// TIA Portal V17 export
// export: Created 2024-09-02T21:27:54.0688981Z, ExportSetting WithDefaults, DisplayName Totally Integrated Automation Portal, DisplayVersion V17 Update 7, DisplayName TIA Portal Openness, DisplayVersion V17 Update 7, DisplayName TIA Portal Version Control Interface, DisplayVersion V17, DisplayName SINAMICS Startdrive Advanced, DisplayVersion V17 SP2, DisplayName SINAMICS Startdrive G110M, G120, G120C, G120D, G120P, G115D, DisplayVersion V17 SP2, DisplayName SINAMICS Startdrive G130, G150, S120, S150, SINAMICS MV, S210, DisplayVersion V17 SP2, DisplayName STEP 7 Professional, DisplayVersion V17 Update 7, DisplayName STEP 7 Safety, DisplayVersion V17 Update 6, DisplayName WinCC Advanced / Unified PC, DisplayVersion V17 Update 7
FUNCTION "inputsMapping" : Void   // FC1, LAD
{ S7_Optimized_Access := 'TRUE' }
VERSION : 0.1
// stored: AutoNumber true, IsIECCheckEnabled false, SetENOAutomatically false, UDAEnableTagReadback false
BEGIN

REGION Network 1: A00.- Clear Data
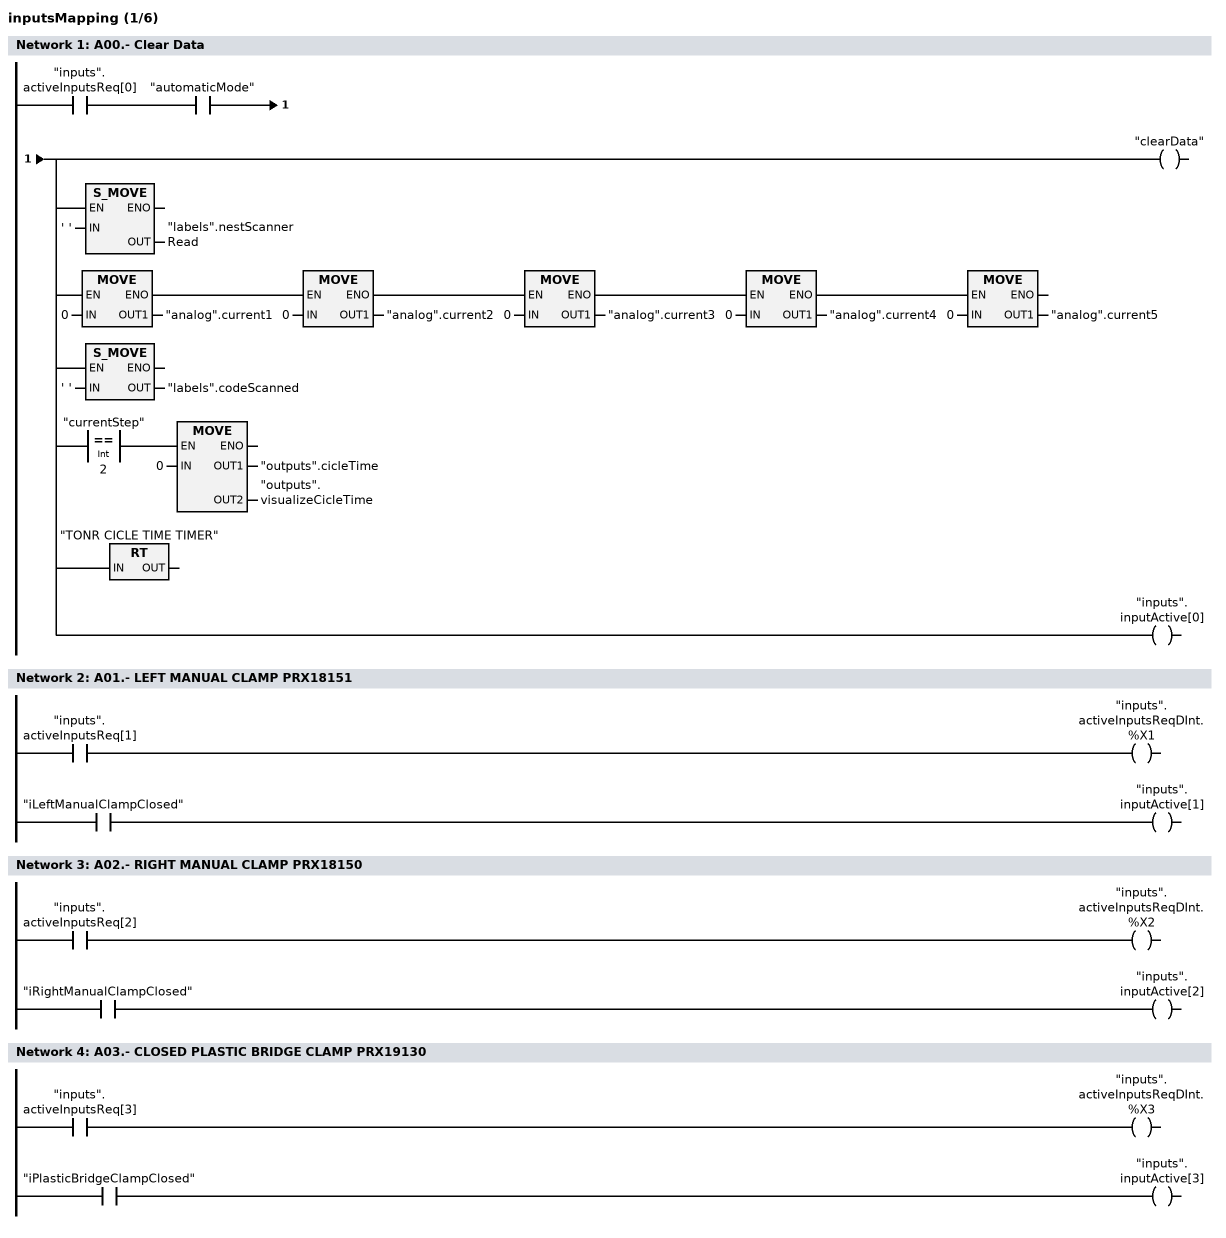
   RUNG wire#powerrail
      Contact( "inputs".activeInputsReq[0] )
      Contact( "automaticMode" )
      wire#w1
      Coil( "clearData" )
   END_RUNG
   RUNG wire#w1
      S_Move(in := ' ', out => "labels".nestScannerRead)
   END_RUNG
   RUNG wire#w1
      Move(in := 0, out1 => "analog".current1)
      Move(in := 0, out1 => "analog".current2)
      Move(in := 0, out1 => "analog".current3)
      Move(in := 0, out1 => "analog".current4)
      Move(in := 0, out1 => "analog".current5)
   END_RUNG
   RUNG wire#w1
      S_Move(in := ' ', out => "labels".codeScanned)
   END_RUNG
   RUNG wire#w1
      { S7_Templates := "SrcType := Int" } EQ_Contact(in1 := "currentStep", in2 := 2)
      Move(in := 0, out1 => "outputs".cicleTime, out2 => "outputs".visualizeCicleTime)
   END_RUNG
   RUNG wire#w1
      RT_Coil( "TONR CICLE TIME TIMER" )
   END_RUNG
   RUNG wire#w1
      Coil( "inputs".inputActive[0] )
   END_RUNG
   // the same network as SCL:
   "clearData" := "inputs".activeInputsReq[0] AND "automaticMode";
   IF "clearData" THEN
       "labels".nestScannerRead := ' ';
       "analog".current1 := 0;
       "analog".current2 := 0;
       "analog".current3 := 0;
       "analog".current4 := 0;
       "analog".current5 := 0;
       "labels".codeScanned := ' ';
   END_IF;
   IF "clearData" AND ("currentStep" = 2) THEN
       "outputs".cicleTime := 0;
       "outputs".visualizeCicleTime := 0;
   END_IF;
   IF "clearData" THEN RESET_TIMER("TONR CICLE TIME TIMER"); END_IF;
   "inputs".inputActive[0] := "clearData";
END_REGION

REGION Network 2: A01.- LEFT MANUAL CLAMP PRX18151
   RUNG wire#powerrail
      Contact( "inputs".activeInputsReq[1] )
      Coil( "inputs".activeInputsReqDInt.%X1 )
   END_RUNG
   RUNG wire#powerrail
      Contact( "iLeftManualClampClosed" )
      Coil( "inputs".inputActive[1] )
   END_RUNG
   // the same network as SCL:
   "inputs".activeInputsReqDInt.%X1 := "inputs".activeInputsReq[1];
   "inputs".inputActive[1] := "iLeftManualClampClosed";
END_REGION

REGION Network 3: A02.- RIGHT MANUAL CLAMP PRX18150
   RUNG wire#powerrail
      Contact( "inputs".activeInputsReq[2] )
      Coil( "inputs".activeInputsReqDInt.%X2 )
   END_RUNG
   RUNG wire#powerrail
      Contact( "iRightManualClampClosed" )
      Coil( "inputs".inputActive[2] )
   END_RUNG
   // the same network as SCL:
   "inputs".activeInputsReqDInt.%X2 := "inputs".activeInputsReq[2];
   "inputs".inputActive[2] := "iRightManualClampClosed";
END_REGION

REGION Network 4: A03.- CLOSED PLASTIC BRIDGE CLAMP PRX19130
   RUNG wire#powerrail
      Contact( "inputs".activeInputsReq[3] )
      Coil( "inputs".activeInputsReqDInt.%X3 )
   END_RUNG
   RUNG wire#powerrail
      Contact( "iPlasticBridgeClampClosed" )
      Coil( "inputs".inputActive[3] )
   END_RUNG
   // the same network as SCL:
   "inputs".activeInputsReqDInt.%X3 := "inputs".activeInputsReq[3];
   "inputs".inputActive[3] := "iPlasticBridgeClampClosed";
END_REGION

REGION Network 5: A04.- PLASTIC BRIDGE PRESENT PRX19090
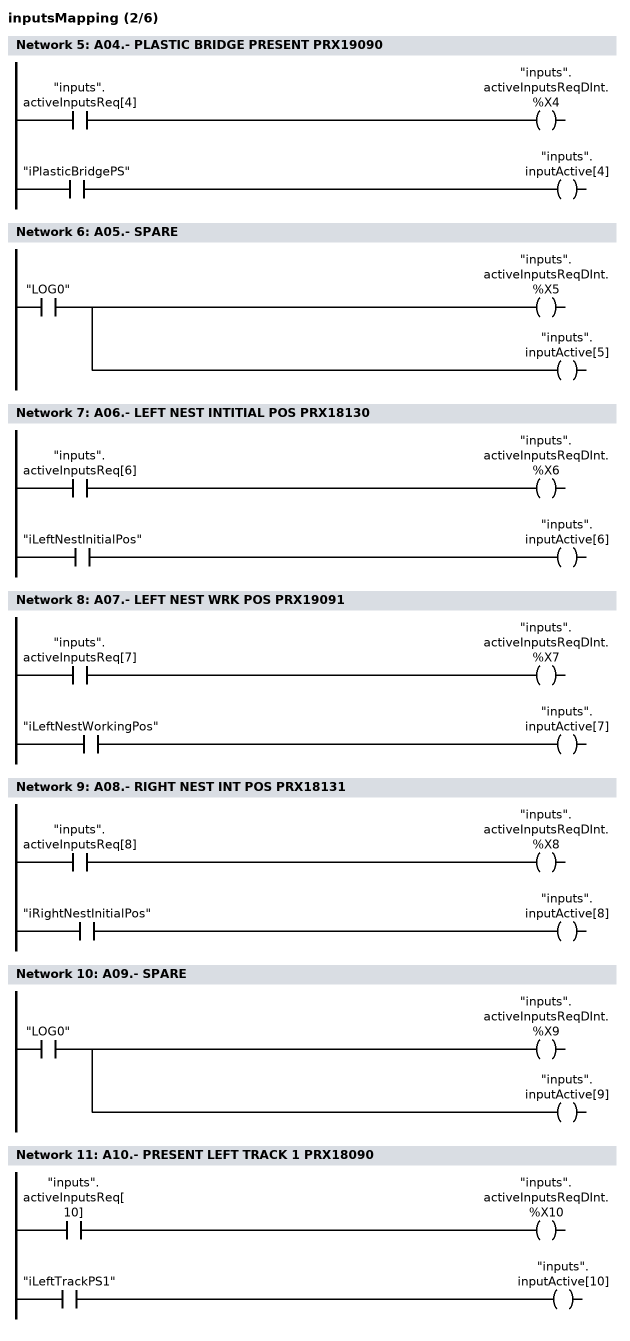
   RUNG wire#powerrail
      Contact( "inputs".activeInputsReq[4] )
      Coil( "inputs".activeInputsReqDInt.%X4 )
   END_RUNG
   RUNG wire#powerrail
      Contact( "iPlasticBridgePS" )
      Coil( "inputs".inputActive[4] )
   END_RUNG
   // the same network as SCL:
   "inputs".activeInputsReqDInt.%X4 := "inputs".activeInputsReq[4];
   "inputs".inputActive[4] := "iPlasticBridgePS";
END_REGION

REGION Network 6: A05.- SPARE
   RUNG wire#powerrail
      Contact( "LOG0" )
      wire#w1
      Coil( "inputs".activeInputsReqDInt.%X5 )
   END_RUNG
   RUNG wire#w1
      Coil( "inputs".inputActive[5] )
   END_RUNG
   // the same network as SCL:
   "inputs".activeInputsReqDInt.%X5 := "LOG0";
   "inputs".inputActive[5] := "LOG0";
END_REGION

REGION Network 7: A06.- LEFT NEST INTITIAL POS PRX18130
   RUNG wire#powerrail
      Contact( "inputs".activeInputsReq[6] )
      Coil( "inputs".activeInputsReqDInt.%X6 )
   END_RUNG
   RUNG wire#powerrail
      Contact( "iLeftNestInitialPos" )
      Coil( "inputs".inputActive[6] )
   END_RUNG
   // the same network as SCL:
   "inputs".activeInputsReqDInt.%X6 := "inputs".activeInputsReq[6];
   "inputs".inputActive[6] := "iLeftNestInitialPos";
END_REGION

REGION Network 8: A07.- LEFT NEST WRK POS PRX19091
   RUNG wire#powerrail
      Contact( "inputs".activeInputsReq[7] )
      Coil( "inputs".activeInputsReqDInt.%X7 )
   END_RUNG
   RUNG wire#powerrail
      Contact( "iLeftNestWorkingPos" )
      Coil( "inputs".inputActive[7] )
   END_RUNG
   // the same network as SCL:
   "inputs".activeInputsReqDInt.%X7 := "inputs".activeInputsReq[7];
   "inputs".inputActive[7] := "iLeftNestWorkingPos";
END_REGION

REGION Network 9: A08.- RIGHT NEST INT POS PRX18131
   RUNG wire#powerrail
      Contact( "inputs".activeInputsReq[8] )
      Coil( "inputs".activeInputsReqDInt.%X8 )
   END_RUNG
   RUNG wire#powerrail
      Contact( "iRightNestInitialPos" )
      Coil( "inputs".inputActive[8] )
   END_RUNG
   // the same network as SCL:
   "inputs".activeInputsReqDInt.%X8 := "inputs".activeInputsReq[8];
   "inputs".inputActive[8] := "iRightNestInitialPos";
END_REGION

REGION Network 10: A09.- SPARE
   RUNG wire#powerrail
      Contact( "LOG0" )
      wire#w1
      Coil( "inputs".activeInputsReqDInt.%X9 )
   END_RUNG
   RUNG wire#w1
      Coil( "inputs".inputActive[9] )
   END_RUNG
   // the same network as SCL:
   "inputs".activeInputsReqDInt.%X9 := "LOG0";
   "inputs".inputActive[9] := "LOG0";
END_REGION

REGION Network 11: A10.- PRESENT LEFT TRACK 1 PRX18090
   RUNG wire#powerrail
      Contact( "inputs".activeInputsReq[10] )
      Coil( "inputs".activeInputsReqDInt.%X10 )
   END_RUNG
   RUNG wire#powerrail
      Contact( "iLeftTrackPS1" )
      Coil( "inputs".inputActive[10] )
   END_RUNG
   // the same network as SCL:
   "inputs".activeInputsReqDInt.%X10 := "inputs".activeInputsReq[10];
   "inputs".inputActive[10] := "iLeftTrackPS1";
END_REGION

REGION Network 12: A11.- PRESENT RIGHT TRACK 1 PRX18110
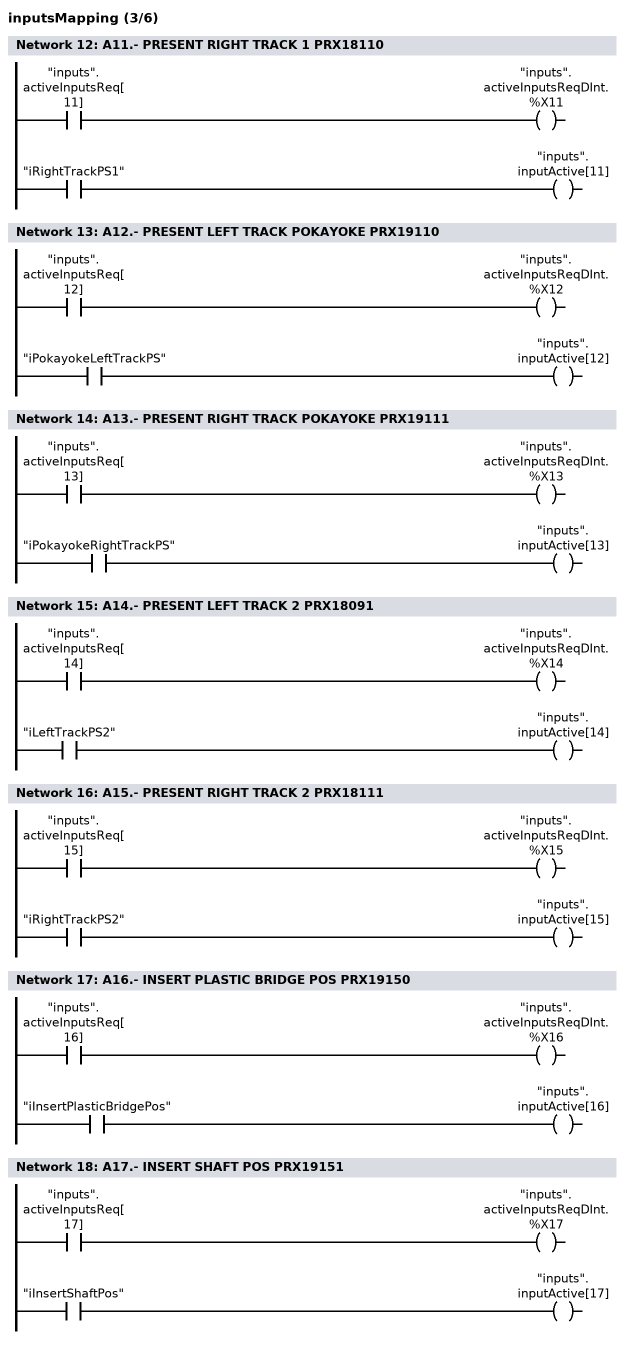
   RUNG wire#powerrail
      Contact( "inputs".activeInputsReq[11] )
      Coil( "inputs".activeInputsReqDInt.%X11 )
   END_RUNG
   RUNG wire#powerrail
      Contact( "iRightTrackPS1" )
      Coil( "inputs".inputActive[11] )
   END_RUNG
   // the same network as SCL:
   "inputs".activeInputsReqDInt.%X11 := "inputs".activeInputsReq[11];
   "inputs".inputActive[11] := "iRightTrackPS1";
END_REGION

REGION Network 13: A12.- PRESENT LEFT TRACK POKAYOKE PRX19110
   RUNG wire#powerrail
      Contact( "inputs".activeInputsReq[12] )
      Coil( "inputs".activeInputsReqDInt.%X12 )
   END_RUNG
   RUNG wire#powerrail
      Contact( "iPokayokeLeftTrackPS" )
      Coil( "inputs".inputActive[12] )
   END_RUNG
   // the same network as SCL:
   "inputs".activeInputsReqDInt.%X12 := "inputs".activeInputsReq[12];
   "inputs".inputActive[12] := "iPokayokeLeftTrackPS";
END_REGION

REGION Network 14: A13.- PRESENT RIGHT TRACK POKAYOKE PRX19111
   RUNG wire#powerrail
      Contact( "inputs".activeInputsReq[13] )
      Coil( "inputs".activeInputsReqDInt.%X13 )
   END_RUNG
   RUNG wire#powerrail
      Contact( "iPokayokeRightTrackPS" )
      Coil( "inputs".inputActive[13] )
   END_RUNG
   // the same network as SCL:
   "inputs".activeInputsReqDInt.%X13 := "inputs".activeInputsReq[13];
   "inputs".inputActive[13] := "iPokayokeRightTrackPS";
END_REGION

REGION Network 15: A14.- PRESENT LEFT TRACK 2 PRX18091
   RUNG wire#powerrail
      Contact( "inputs".activeInputsReq[14] )
      Coil( "inputs".activeInputsReqDInt.%X14 )
   END_RUNG
   RUNG wire#powerrail
      Contact( "iLeftTrackPS2" )
      Coil( "inputs".inputActive[14] )
   END_RUNG
   // the same network as SCL:
   "inputs".activeInputsReqDInt.%X14 := "inputs".activeInputsReq[14];
   "inputs".inputActive[14] := "iLeftTrackPS2";
END_REGION

REGION Network 16: A15.- PRESENT RIGHT TRACK 2 PRX18111
   RUNG wire#powerrail
      Contact( "inputs".activeInputsReq[15] )
      Coil( "inputs".activeInputsReqDInt.%X15 )
   END_RUNG
   RUNG wire#powerrail
      Contact( "iRightTrackPS2" )
      Coil( "inputs".inputActive[15] )
   END_RUNG
   // the same network as SCL:
   "inputs".activeInputsReqDInt.%X15 := "inputs".activeInputsReq[15];
   "inputs".inputActive[15] := "iRightTrackPS2";
END_REGION

REGION Network 17: A16.- INSERT PLASTIC BRIDGE POS PRX19150
   RUNG wire#powerrail
      Contact( "inputs".activeInputsReq[16] )
      Coil( "inputs".activeInputsReqDInt.%X16 )
   END_RUNG
   RUNG wire#powerrail
      Contact( "iInsertPlasticBridgePos" )
      Coil( "inputs".inputActive[16] )
   END_RUNG
   // the same network as SCL:
   "inputs".activeInputsReqDInt.%X16 := "inputs".activeInputsReq[16];
   "inputs".inputActive[16] := "iInsertPlasticBridgePos";
END_REGION

REGION Network 18: A17.- INSERT SHAFT POS PRX19151
   RUNG wire#powerrail
      Contact( "inputs".activeInputsReq[17] )
      Coil( "inputs".activeInputsReqDInt.%X17 )
   END_RUNG
   RUNG wire#powerrail
      Contact( "iInsertShaftPos" )
      Coil( "inputs".inputActive[17] )
   END_RUNG
   // the same network as SCL:
   "inputs".activeInputsReqDInt.%X17 := "inputs".activeInputsReq[17];
   "inputs".inputActive[17] := "iInsertShaftPos";
END_REGION

REGION Network 19: A18.- REMOVE PIECE
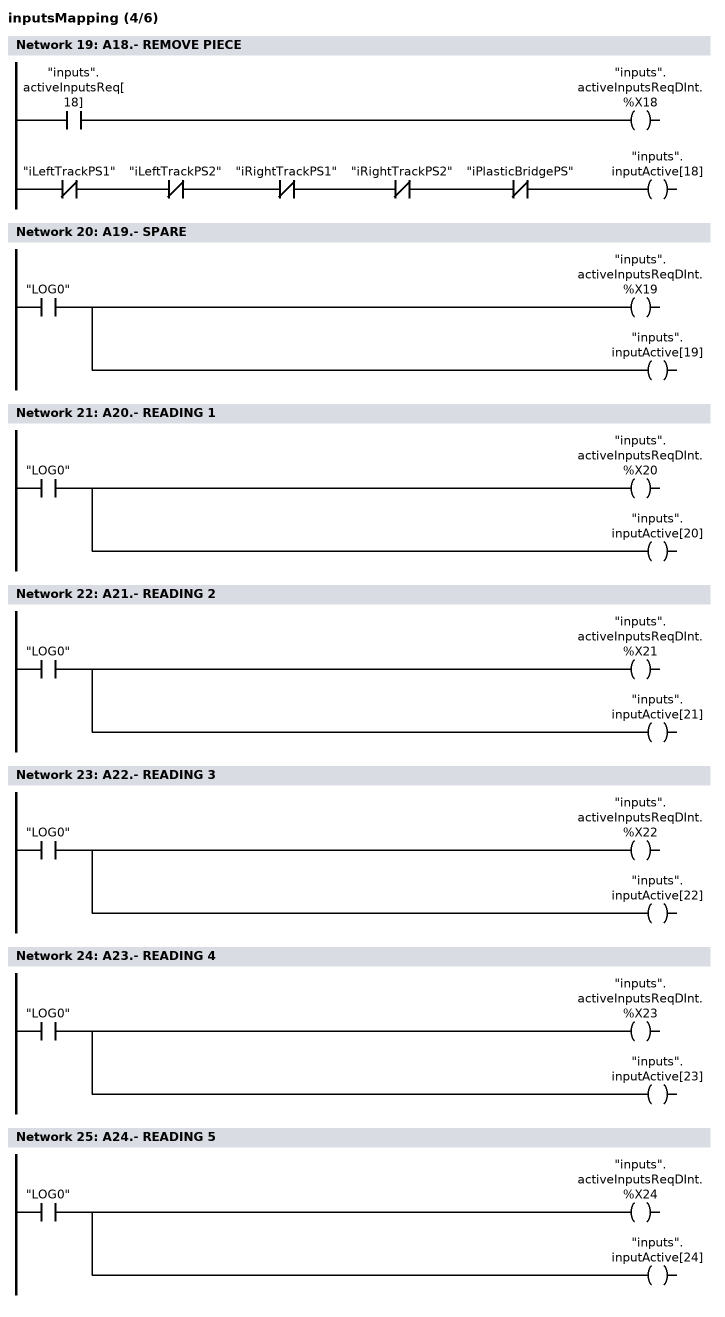
   RUNG wire#powerrail
      Contact( "inputs".activeInputsReq[18] )
      Coil( "inputs".activeInputsReqDInt.%X18 )
   END_RUNG
   RUNG wire#powerrail
      I_Contact( "iLeftTrackPS1" )
      I_Contact( "iLeftTrackPS2" )
      I_Contact( "iRightTrackPS1" )
      I_Contact( "iRightTrackPS2" )
      I_Contact( "iPlasticBridgePS" )
      Coil( "inputs".inputActive[18] )
   END_RUNG
   // the same network as SCL:
   "inputs".activeInputsReqDInt.%X18 := "inputs".activeInputsReq[18];
   "inputs".inputActive[18] := NOT "iLeftTrackPS1" AND NOT "iLeftTrackPS2" AND NOT "iRightTrackPS1" AND NOT "iRightTrackPS2" AND NOT "iPlasticBridgePS";
END_REGION

REGION Network 20: A19.- SPARE
   RUNG wire#powerrail
      Contact( "LOG0" )
      wire#w1
      Coil( "inputs".activeInputsReqDInt.%X19 )
   END_RUNG
   RUNG wire#w1
      Coil( "inputs".inputActive[19] )
   END_RUNG
   // the same network as SCL:
   "inputs".activeInputsReqDInt.%X19 := "LOG0";
   "inputs".inputActive[19] := "LOG0";
END_REGION

REGION Network 21: A20.- READING 1
   RUNG wire#powerrail
      Contact( "LOG0" )
      wire#w1
      Coil( "inputs".activeInputsReqDInt.%X20 )
   END_RUNG
   RUNG wire#w1
      Coil( "inputs".inputActive[20] )
   END_RUNG
   // the same network as SCL:
   "inputs".activeInputsReqDInt.%X20 := "LOG0";
   "inputs".inputActive[20] := "LOG0";
END_REGION

REGION Network 22: A21.- READING 2
   RUNG wire#powerrail
      Contact( "LOG0" )
      wire#w1
      Coil( "inputs".activeInputsReqDInt.%X21 )
   END_RUNG
   RUNG wire#w1
      Coil( "inputs".inputActive[21] )
   END_RUNG
   // the same network as SCL:
   "inputs".activeInputsReqDInt.%X21 := "LOG0";
   "inputs".inputActive[21] := "LOG0";
END_REGION

REGION Network 23: A22.- READING 3
   RUNG wire#powerrail
      Contact( "LOG0" )
      wire#w1
      Coil( "inputs".activeInputsReqDInt.%X22 )
   END_RUNG
   RUNG wire#w1
      Coil( "inputs".inputActive[22] )
   END_RUNG
   // the same network as SCL:
   "inputs".activeInputsReqDInt.%X22 := "LOG0";
   "inputs".inputActive[22] := "LOG0";
END_REGION

REGION Network 24: A23.- READING 4
   RUNG wire#powerrail
      Contact( "LOG0" )
      wire#w1
      Coil( "inputs".activeInputsReqDInt.%X23 )
   END_RUNG
   RUNG wire#w1
      Coil( "inputs".inputActive[23] )
   END_RUNG
   // the same network as SCL:
   "inputs".activeInputsReqDInt.%X23 := "LOG0";
   "inputs".inputActive[23] := "LOG0";
END_REGION

REGION Network 25: A24.- READING 5
   RUNG wire#powerrail
      Contact( "LOG0" )
      wire#w1
      Coil( "inputs".activeInputsReqDInt.%X24 )
   END_RUNG
   RUNG wire#w1
      Coil( "inputs".inputActive[24] )
   END_RUNG
   // the same network as SCL:
   "inputs".activeInputsReqDInt.%X24 := "LOG0";
   "inputs".inputActive[24] := "LOG0";
END_REGION

REGION Network 26: A25.- SPARE
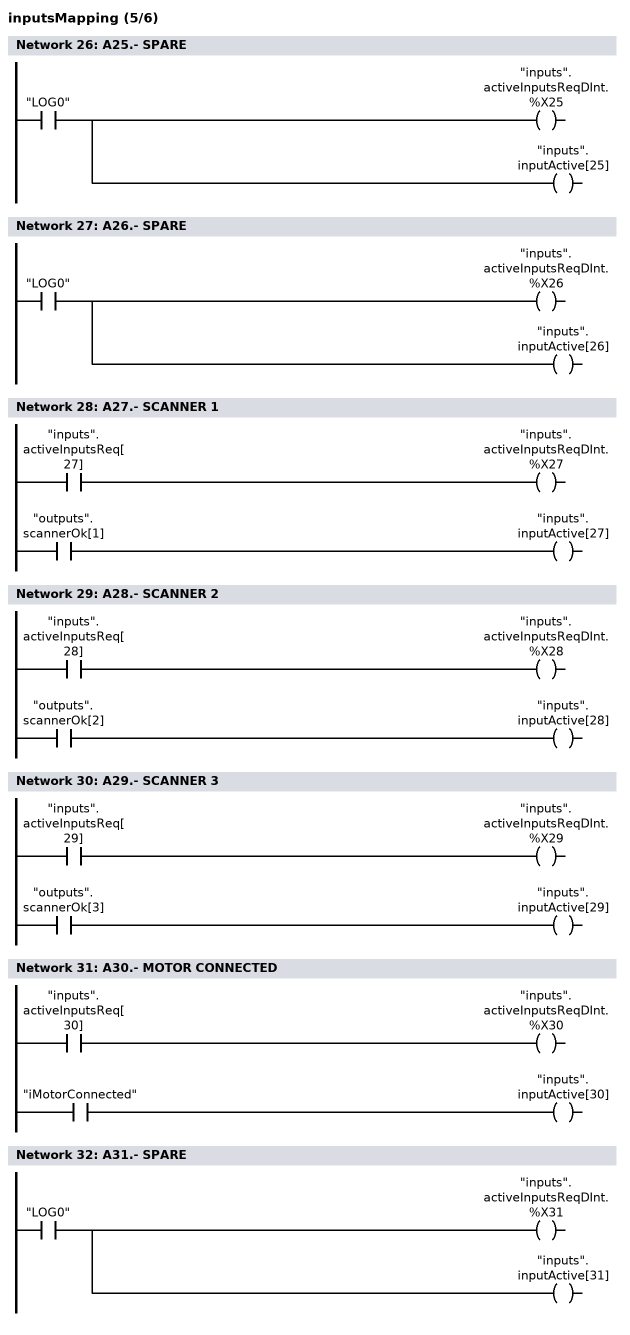
   RUNG wire#powerrail
      Contact( "LOG0" )
      wire#w1
      Coil( "inputs".activeInputsReqDInt.%X25 )
   END_RUNG
   RUNG wire#w1
      Coil( "inputs".inputActive[25] )
   END_RUNG
   // the same network as SCL:
   "inputs".activeInputsReqDInt.%X25 := "LOG0";
   "inputs".inputActive[25] := "LOG0";
END_REGION

REGION Network 27: A26.- SPARE
   RUNG wire#powerrail
      Contact( "LOG0" )
      wire#w1
      Coil( "inputs".activeInputsReqDInt.%X26 )
   END_RUNG
   RUNG wire#w1
      Coil( "inputs".inputActive[26] )
   END_RUNG
   // the same network as SCL:
   "inputs".activeInputsReqDInt.%X26 := "LOG0";
   "inputs".inputActive[26] := "LOG0";
END_REGION

REGION Network 28: A27.- SCANNER 1
   RUNG wire#powerrail
      Contact( "inputs".activeInputsReq[27] )
      Coil( "inputs".activeInputsReqDInt.%X27 )
   END_RUNG
   RUNG wire#powerrail
      Contact( "outputs".scannerOk[1] )
      Coil( "inputs".inputActive[27] )
   END_RUNG
   // the same network as SCL:
   "inputs".activeInputsReqDInt.%X27 := "inputs".activeInputsReq[27];
   "inputs".inputActive[27] := "outputs".scannerOk[1];
END_REGION

REGION Network 29: A28.- SCANNER 2
   RUNG wire#powerrail
      Contact( "inputs".activeInputsReq[28] )
      Coil( "inputs".activeInputsReqDInt.%X28 )
   END_RUNG
   RUNG wire#powerrail
      Contact( "outputs".scannerOk[2] )
      Coil( "inputs".inputActive[28] )
   END_RUNG
   // the same network as SCL:
   "inputs".activeInputsReqDInt.%X28 := "inputs".activeInputsReq[28];
   "inputs".inputActive[28] := "outputs".scannerOk[2];
END_REGION

REGION Network 30: A29.- SCANNER 3
   RUNG wire#powerrail
      Contact( "inputs".activeInputsReq[29] )
      Coil( "inputs".activeInputsReqDInt.%X29 )
   END_RUNG
   RUNG wire#powerrail
      Contact( "outputs".scannerOk[3] )
      Coil( "inputs".inputActive[29] )
   END_RUNG
   // the same network as SCL:
   "inputs".activeInputsReqDInt.%X29 := "inputs".activeInputsReq[29];
   "inputs".inputActive[29] := "outputs".scannerOk[3];
END_REGION

REGION Network 31: A30.- MOTOR CONNECTED
   RUNG wire#powerrail
      Contact( "inputs".activeInputsReq[30] )
      Coil( "inputs".activeInputsReqDInt.%X30 )
   END_RUNG
   RUNG wire#powerrail
      Contact( "iMotorConnected" )
      Coil( "inputs".inputActive[30] )
   END_RUNG
   // the same network as SCL:
   "inputs".activeInputsReqDInt.%X30 := "inputs".activeInputsReq[30];
   "inputs".inputActive[30] := "iMotorConnected";
END_REGION

REGION Network 32: A31.- SPARE
   RUNG wire#powerrail
      Contact( "LOG0" )
      wire#w1
      Coil( "inputs".activeInputsReqDInt.%X31 )
   END_RUNG
   RUNG wire#w1
      Coil( "inputs".inputActive[31] )
   END_RUNG
   // the same network as SCL:
   "inputs".activeInputsReqDInt.%X31 := "LOG0";
   "inputs".inputActive[31] := "LOG0";
END_REGION

REGION Network 33: HMI SENSOR OVERVIEW
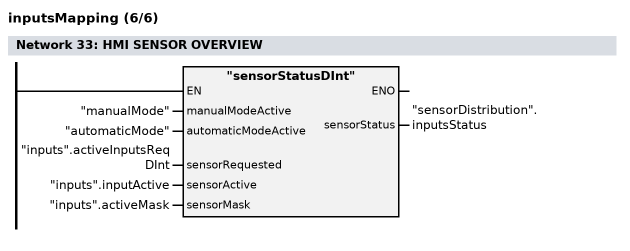
   RUNG wire#powerrail
      "sensorStatusDInt"(manualModeActive := "manualMode", automaticModeActive := "automaticMode", sensorRequested := "inputs".activeInputsReqDInt, sensorActive := "inputs".inputActive, sensorMask := "inputs".activeMask, sensorStatus => "sensorDistribution".inputsStatus)
   END_RUNG
   // the same network as SCL:
   "sensorStatusDInt"(manualModeActive := "manualMode",
                      automaticModeActive := "automaticMode",
                      sensorRequested := "inputs".activeInputsReqDInt,
                      sensorActive := "inputs".inputActive,
                      sensorMask := "inputs".activeMask,
                      sensorStatus => "sensorDistribution".inputsStatus);
END_REGION
END_FUNCTION
